(* IEC 61131-3 sources: SIGMATEK-Jumag-Utils-Examples/formulasSteam/Class/antoineFormular, 1 file *)

(* ---- antoineFormular.st ---- *)
(*!
<Class
	Name               = "antoineFormular"
	Revision           = "0.0"
	RealtimeTask       = "false"
	CyclicTask         = "true"
	DefCyclictime      = "100 ms"
	BackgroundTask     = "false"
	Sigmatek           = "false"
	OSInterface        = "false"
	HighPriority       = "false"
	Automatic          = "false"
	UpdateMode         = "Prescan"
	SharedCommandTable = "true"
	Objectsize         = "(624,120)">
	<Channels>
		<Server Name="antoinePressure" Visualized="false" Initialize="false" WriteProtected="true" Retentive="false"/>
		<Server Name="antoineTemperature" Visualized="false" Initialize="false" WriteProtected="true" Retentive="false"/>
		<Server Name="ClassSvr" Visualized="false" Initialize="false" WriteProtected="true" Retentive="false"/>
		<Client Name="pressure" Required="true" Internal="false"/>
	</Channels>
	<Dependencies>
		<Files>
			<File Path=".\Source\formulasSteam.c"/>
		</Files>
	</Dependencies>
</Class>
*)
antoineFormular : CLASS
  //Servers:
	ClassSvr 	: SvrChCmd_DINT;
	antoineTemperature 	: SvrCh_REAL;
	antoinePressure 	: SvrCh_REAL;
  //Clients:
	pressure 	: CltCh_DINT;
  //Variables:
  //Functions:

	FUNCTION VIRTUAL GLOBAL CyWork
		VAR_INPUT
			EAX 	: UDINT;
		END_VAR
		VAR_OUTPUT
			state (EAX) 	: UDINT;
		END_VAR;
  //Tables:
	FUNCTION @STD
		VAR_OUTPUT
			ret_code	: CONFSTATES;
		END_VAR;
	FUNCTION GLOBAL TAB @CT_;
END_CLASS;

Function Global __cdecl antoineFormT
VAR_INPUT
  INPUT : REAL;
  OPTION : BOOL;
END_VAR
VAR_OUTPUT
  Q : REAL;
END_VAR;

Function Global __cdecl antoineFormP
VAR_INPUT
  INPUT : REAL;
END_VAR
VAR_OUTPUT
  Q : REAL;
END_VAR;

FUNCTION VIRTUAL GLOBAL antoineFormular::CyWork
	VAR_INPUT
		EAX 	: UDINT;
	END_VAR
	VAR_OUTPUT
		state (EAX) 	: UDINT;
	END_VAR

  pressure := pressure.Read();

  antoineTemperature := antoineFormT(INPUT:= to_real(pressure),OPTION:= TRUE );

  antoinePressure := antoineFormP(INPUT:=antoineTemperature);

	state := READY;

END_FUNCTION
